VAR_GLOBAL
	RxBufferEL			: ComBuffer;	(* Receive data buffer; used with all receive function blocks *)
	TxBufferEL			: ComBuffer;	(* Transmit data buffer; used with all receive function blocks *)
END_VAR

(* stored: Version 1.1.0.1, ProductVersion 3.1.4024.12
   GVL GVL: Id {3e4349e6-a99a-4aa8-b94a-96e30307ccae} *)
